# EPICS autosave request: calcApp/Db/userCalcGlobalEnable_settings.req
$(P)userCalcGlobalEnable
